PROGRAM myCNC_CureQue
VAR
END_VAR

END_PROGRAM

(* stored: Version 1.1.0.1, ProductVersion 3.1.4024.11
   POU myCNC_CureQue: Id {8ee457db-f410-4e86-82d6-a405a74cff8d}, SpecialFunc None *)
